Staubli VAL3: onExit.pgx

program onExit()
begin
  // on EXIT
  //
  if cycleStatus:bSimulation
    call stopCycle()
  endIf
  // clean the movement
  if !isEmpty()
    resetMotion()
  endIf
  call use:nullKey(nKey)
  taskKill("stepping")
end
